(* CoDeSys 2.3.9.41 project: Mixer2_v1.pro *)
(* Libraries: Standard.lib 4.10.05 11:14:46, IecSfc.lib 13.4.06 15:51:28, SYSLIBCALLBACK.LIB 26.9.08 16:43:52 *)

(* Task configuration *)
TASK NewTask (PRIORITY := 1); (* freewheeling *)
	VIS_PRG();
	PLC_PRG();
END_TASK

(* POU VIS_PRG, ST *)
PROGRAM VIS_PRG
VAR
END_VAR

END_PROGRAM

(* POU PLC_PRG, ST *)
PROGRAM PLC_PRG
VAR
END_VAR

END_PROGRAM

(* Visualisation Vis_Mixer2
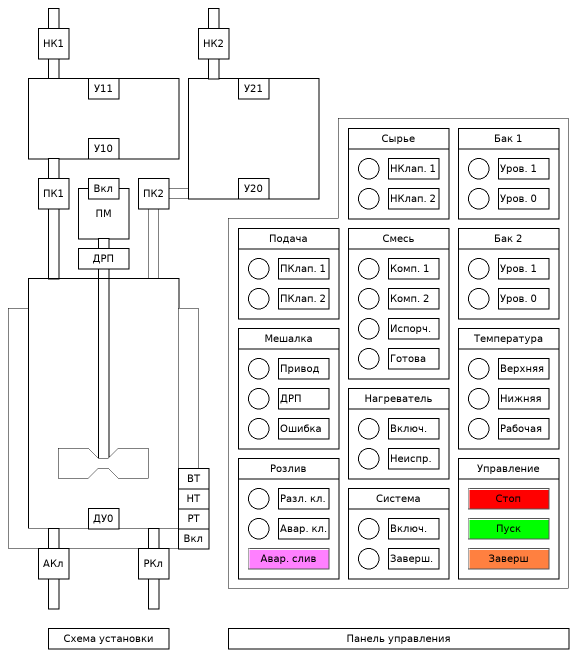
rectangle at (250,50)-(281,81): text "НК2"
rectangle at (90,50)-(121,81): text "НК1"
rectangle at (130,210)-(181,261): text "ПМ"
rectangle at (140,200)-(171,221): text "Вкл"
rectangle at (130,270)-(181,291): text "ДРП"
rectangle at (190,200)-(221,231): text "ПК2"
rectangle at (140,100)-(171,121): text "У11"
rectangle at (140,160)-(171,181): text "У10"
rectangle at (290,100)-(321,121): text "У21"
rectangle at (290,200)-(321,221): text "У20"
rectangle at (140,530)-(171,551): text "ДУ0"
rectangle at (230,550)-(261,571): text "Вкл"
rectangle at (230,530)-(261,551): text "РТ"
rectangle at (230,510)-(261,531): text "НТ"
rectangle at (230,490)-(261,511): text "ВТ"
rectangle at (90,570)-(121,601): text "АКл"
rectangle at (190,570)-(221,601): text "РКл"
button at (300,570)-(381,591): text "Авар. слив"
rectangle at (330,540)-(381,561): text "Авар. кл."
rectangle at (330,510)-(381,531): text "Разл. кл."
rectangle at (290,480)-(391,501): text "Розлив"
rectangle at (440,570)-(491,591): text "Заверш."
rectangle at (440,540)-(491,561): text "Включ."
rectangle at (400,510)-(501,531): text "Система"
rectangle at (440,470)-(491,491): text "Неиспр."
rectangle at (440,440)-(491,461): text "Включ."
rectangle at (400,410)-(501,431): text "Нагреватель"
rectangle at (330,440)-(381,461): text "Ошибка"
rectangle at (330,410)-(381,431): text "ДРП"
rectangle at (330,380)-(381,401): text "Привод"
rectangle at (290,350)-(391,371): text "Мешалка"
rectangle at (330,310)-(381,331): text "ПКлап. 2"
rectangle at (330,280)-(381,301): text "ПКлап. 1"
rectangle at (290,250)-(391,271): text "Подача"
rectangle at (440,370)-(491,391): text "Готова"
rectangle at (440,340)-(491,361): text "Испорч."
rectangle at (440,310)-(491,331): text "Комп. 2"
rectangle at (440,280)-(491,301): text "Комп. 1"
rectangle at (400,250)-(501,271): text "Смесь"
button at (520,570)-(601,591): text "Заверш"
button at (520,540)-(601,561): text "Пуск"
button at (520,510)-(601,531): text "Стоп"
rectangle at (510,480)-(611,501): text "Управление"
rectangle at (550,440)-(601,461): text "Рабочая"
rectangle at (550,410)-(601,431): text "Нижняя"
rectangle at (550,380)-(601,401): text "Верхняя"
rectangle at (510,350)-(611,371): text "Температура"
rectangle at (550,310)-(601,331): text "Уров. 0"
rectangle at (550,280)-(601,301): text "Уров. 1"
rectangle at (510,250)-(611,271): text "Бак 2"
rectangle at (550,210)-(601,231): text "Уров. 0"
rectangle at (550,180)-(601,201): text "Уров. 1"
rectangle at (510,150)-(611,171): text "Бак 1"
rectangle at (440,210)-(491,231): text "НКлап. 2"
rectangle at (440,180)-(491,201): text "НКлап. 1"
rectangle at (400,150)-(501,171): text "Сырье"
rectangle at (90,200)-(121,231): text "ПК1"
rectangle at (100,650)-(221,671): text "Схема установки"
rectangle at (280,650)-(621,671): text "Панель управления"
49 more shapes without text or variables
*)
